{attribute 'qualified_only'}
{attribute 'strict'}
{attribute 'to_string'}
TYPE ProcessExec_e :
(
	StartImmediately,
	StartSynchronize,
	_MAX
);
END_TYPE

(* stored: Version 1.1.0.1, ProductVersion 3.1.4024.6
   DUT ProcessExec_e: Id {23a6662d-9144-4a13-83a7-1227e92b8661} *)
